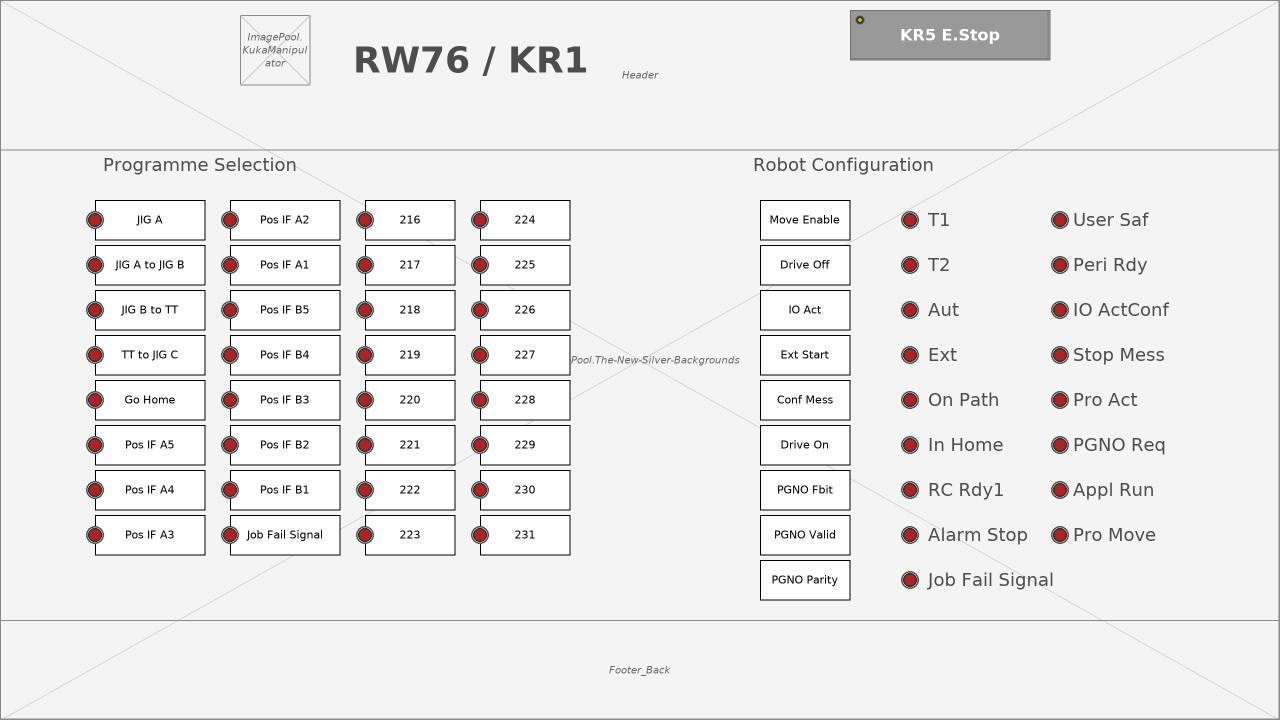
VISUALIZATION PAGE_KR5  // 1280x720
    Image (0,0 1280x720), image: ImagePool.The-New-Silver-Backgrounds
    Frame (0,620 1280x100)
        shows Footer_Back()
    Frame (0,0 1280x150)
        shows Header()
    Label (350,40 300x40), "RW76 / KR1"
    Label (100,150 200x30), "Programme Selection"
    Label (750,150 200x30), "Robot Configuration"
    Lamp1 (900,210 20x20), variable: KR5.bInBit[1,0], style: Lamp-Lamp1-Red
    Lamp1 (900,255 20x20), variable: KR5.bInBit[1,1], style: Lamp-Lamp1-Red
    Lamp1 (900,300 20x20), variable: KR5.bInBit[1,2], style: Lamp-Lamp1-Red
    Lamp1 (900,345 20x20), variable: KR5.bInBit[1,3], style: Lamp-Lamp1-Red
    Lamp1 (900,390 20x20), variable: KR5.bInBit[1,4], style: Lamp-Lamp1-Red
    Lamp1 (900,435 20x20), variable: KR5.bInBit[1,5], style: Lamp-Lamp1-Red
    Lamp1 (900,480 20x20), variable: KR5.bInBit[1,6], style: Lamp-Lamp1-Red
    Lamp1 (900,525 20x20), variable: KR5.bInBit[1,7], style: Lamp-Lamp1-Red
    Lamp1 (1050,210 20x20), variable: KR5.bInBit[2,0], style: Lamp-Lamp1-Red
    Lamp1 (1050,255 20x20), variable: KR5.bInBit[2,1], style: Lamp-Lamp1-Red
    Lamp1 (1050,300 20x20), variable: KR5.bInBit[2,2], style: Lamp-Lamp1-Red
    Lamp1 (1050,345 20x20), variable: KR5.bInBit[2,3], style: Lamp-Lamp1-Red
    Lamp1 (1050,390 20x20), variable: KR5.bInBit[2,4], style: Lamp-Lamp1-Red
    Lamp1 (1050,435 20x20), variable: KR5.bInBit[2,5], style: Lamp-Lamp1-Red
    Lamp1 (1050,480 20x20), variable: KR5.bInBit[2,6], style: Lamp-Lamp1-Red
    Lamp1 (1050,525 20x20), variable: KR5.bInBit[2,7], style: Lamp-Lamp1-Red
    Group (850,10 200x50)
        Button (0,0 200x50), "KR5 E.Stop"
            toggle KR5.KR5_Estop
        Lamp1 (5,5 10x10), variable: KR5.KR5_Estop, style: Lamp-Lamp1-Yellow
    Image (240,15 70x70), image: ImagePool.KukaManipulator
    RoundedRectangle (760,200 90x40), "Move Enable"
        toggle KR5.bOutBit[1,0]
    RoundedRectangle (760,245 90x40), "Drive Off"
        toggle KR5.bOutBit[1,1]
    RoundedRectangle (760,290 90x40), "IO Act"
        toggle KR5.bOutBit[1,2]
    RoundedRectangle (760,335 90x40), "Ext Start"
        toggle KR5.bOutBit[1,3]
    RoundedRectangle (760,380 90x40), "Conf Mess"
        toggle KR5.bOutBit[1,4]
    RoundedRectangle (760,425 90x40), "Drive On"
        toggle KR5.bOutBit[1,5]
    RoundedRectangle (760,470 90x40), "PGNO Fbit"
        toggle KR5.bOutBit[1,6]
    RoundedRectangle (760,515 90x40), "PGNO Valid"
        toggle KR5.bOutBit[1,7]
    RoundedRectangle (760,560 90x40), "PGNO Parity"
        toggle KR5.bOutBit[2,0]
    RoundedRectangle (95,200 110x40), "JIG A"
        toggle KR5.bOutBit[3,0]
    RoundedRectangle (95,245 110x40), "JIG A to JIG B"
        toggle KR5.bOutBit[3,1]
    RoundedRectangle (95,290 110x40), "JIG B to TT"
        toggle KR5.bOutBit[3,2]
    RoundedRectangle (95,335 110x40), "TT to JIG C"
        toggle KR5.bOutBit[3,3]
    RoundedRectangle (95,380 110x40), "Go Home"
        toggle KR5.bOutBit[3,4]
    RoundedRectangle (95,425 110x40), "Pos IF A5"
        toggle KR5.bOutBit[3,5]
    RoundedRectangle (95,470 110x40), "Pos IF A4"
        toggle KR5.bOutBit[3,6]
    RoundedRectangle (95,515 110x40), "Pos IF A3"
        toggle KR5.bOutBit[3,7]
    Label (1070,205 110x30), "User Saf"
    Label (1070,250 110x30), "Peri Rdy"
    Label (1070,295 110x30), "IO ActConf"
    Label (1070,340 110x30), "Stop Mess"
    Label (1070,385 110x30), "Pro Act"
    Label (1070,430 110x30), "PGNO Req"
    Label (1070,475 110x30), "Appl Run"
    Label (1070,520 110x30), "Pro Move"
    Label (925,205 105x30), "T1"
    Label (925,250 105x30), "T2"
    Label (925,295 105x30), "Aut"
    Label (925,340 105x30), "Ext"
    Label (925,385 105x30), "On Path"
    Label (925,430 105x30), "In Home"
    Label (925,475 105x30), "RC Rdy1"
    Label (925,520 105x30), "Alarm Stop"
    Label (925,565 200x30), "Job Fail Signal"
    Lamp1 (900,570 20x20), variable: KR5.bInBit[4,7], style: Lamp-Lamp1-Red
    RoundedRectangle (230,200 110x40), "Pos IF A2"
        toggle KR5.bOutBit[4,0]
    RoundedRectangle (230,245 110x40), "Pos IF A1"
        toggle KR5.bOutBit[4,1]
    RoundedRectangle (230,290 110x40), "Pos IF B5"
        toggle KR5.bOutBit[4,2]
    RoundedRectangle (230,335 110x40), "Pos IF B4"
        toggle KR5.bOutBit[4,3]
    RoundedRectangle (230,380 110x40), "Pos IF B3"
        toggle KR5.bOutBit[4,4]
    RoundedRectangle (230,425 110x40), "Pos IF B2"
        toggle KR5.bOutBit[4,5]
    RoundedRectangle (230,470 110x40), "Pos IF B1"
        toggle KR5.bOutBit[4,6]
    RoundedRectangle (230,515 110x40), "Job Fail Signal"
        toggle KR5.bOutBit[4,7]
    RoundedRectangle (480,200 90x40), "224"
        toggle KR5.bOutBit[6,0]
    RoundedRectangle (480,245 90x40), "225"
        toggle KR5.bOutBit[6,1]
    RoundedRectangle (480,290 90x40), "226"
        toggle KR5.bOutBit[6,2]
    RoundedRectangle (480,335 90x40), "227"
        toggle KR5.bOutBit[6,3]
    RoundedRectangle (480,380 90x40), "228"
        toggle KR5.bOutBit[6,4]
    RoundedRectangle (480,425 90x40), "229"
        toggle KR5.bOutBit[6,5]
    RoundedRectangle (480,470 90x40), "230"
        toggle KR5.bOutBit[6,6]
    RoundedRectangle (480,515 90x40), "231"
        toggle KR5.bOutBit[6,7]
    Lamp1 (470,210 20x20), variable: KR5.bInBit[6,0], style: Lamp-Lamp1-Red
    Lamp1 (470,255 20x20), variable: KR5.bInBit[6,1], style: Lamp-Lamp1-Red
    Lamp1 (470,300 20x20), variable: KR5.bInBit[6,2], style: Lamp-Lamp1-Red
    Lamp1 (470,345 20x20), variable: KR5.bInBit[6,3], style: Lamp-Lamp1-Red
    Lamp1 (470,390 20x20), variable: KR5.bInBit[6,4], style: Lamp-Lamp1-Red
    Lamp1 (470,435 20x20), variable: KR5.bInBit[6,5], style: Lamp-Lamp1-Red
    Lamp1 (470,480 20x20), variable: KR5.bInBit[6,6], style: Lamp-Lamp1-Red
    Lamp1 (470,525 20x20), variable: KR5.bInBit[6,7], style: Lamp-Lamp1-Red
    RoundedRectangle (365,200 90x40), "216"
        toggle KR5.bOutBit[5,0]
    RoundedRectangle (365,245 90x40), "217"
        toggle KR5.bOutBit[5,1]
    RoundedRectangle (365,290 90x40), "218"
        toggle KR5.bOutBit[5,2]
    RoundedRectangle (365,335 90x40), "219"
        toggle KR5.bOutBit[5,3]
    RoundedRectangle (365,380 90x40), "220"
        toggle KR5.bOutBit[5,4]
    RoundedRectangle (365,425 90x40), "221"
        toggle KR5.bOutBit[5,5]
    RoundedRectangle (365,470 90x40), "222"
        toggle KR5.bOutBit[5,6]
    RoundedRectangle (365,515 90x40), "223"
        toggle KR5.bOutBit[5,7]
    Lamp1 (355,210 20x20), variable: KR5.bInBit[5,0], style: Lamp-Lamp1-Red
    Lamp1 (355,255 20x20), variable: KR5.bInBit[5,1], style: Lamp-Lamp1-Red
    Lamp1 (355,300 20x20), variable: KR5.bInBit[5,2], style: Lamp-Lamp1-Red
    Lamp1 (355,345 20x20), variable: KR5.bInBit[5,3], style: Lamp-Lamp1-Red
    Lamp1 (355,390 20x20), variable: KR5.bInBit[5,4], style: Lamp-Lamp1-Red
    Lamp1 (355,435 20x20), variable: KR5.bInBit[5,5], style: Lamp-Lamp1-Red
    Lamp1 (355,480 20x20), variable: KR5.bInBit[5,6], style: Lamp-Lamp1-Red
    Lamp1 (355,525 20x20), variable: KR5.bInBit[5,7], style: Lamp-Lamp1-Red
    Lamp1 (220,210 20x20), variable: KR5.bInBit[4,0], style: Lamp-Lamp1-Red
    Lamp1 (220,255 20x20), variable: KR5.bInBit[4,1], style: Lamp-Lamp1-Red
    Lamp1 (220,300 20x20), variable: KR5.bInBit[4,2], style: Lamp-Lamp1-Red
    Lamp1 (220,345 20x20), variable: KR5.bInBit[4,3], style: Lamp-Lamp1-Red
    Lamp1 (220,390 20x20), variable: KR5.bInBit[4,4], style: Lamp-Lamp1-Red
    Lamp1 (220,435 20x20), variable: KR5.bInBit[4,5], style: Lamp-Lamp1-Red
    Lamp1 (220,480 20x20), variable: KR5.bInBit[4,6], style: Lamp-Lamp1-Red
    Lamp1 (220,525 20x20), variable: KR5.bInBit[4,7], style: Lamp-Lamp1-Red
    Lamp1 (85,210 20x20), variable: KR5.bInBit[3,0], style: Lamp-Lamp1-Red
    Lamp1 (85,255 20x20), variable: KR5.bInBit[3,1], style: Lamp-Lamp1-Red
    Lamp1 (85,300 20x20), variable: KR5.bInBit[3,2], style: Lamp-Lamp1-Red
    Lamp1 (85,345 20x20), variable: KR5.bInBit[3,3], style: Lamp-Lamp1-Red
    Lamp1 (85,390 20x20), variable: KR5.bInBit[3,4], style: Lamp-Lamp1-Red
    Lamp1 (85,435 20x20), variable: KR5.bInBit[3,5], style: Lamp-Lamp1-Red
    Lamp1 (85,480 20x20), variable: KR5.bInBit[3,6], style: Lamp-Lamp1-Red
    Lamp1 (85,525 20x20), variable: KR5.bInBit[3,7], style: Lamp-Lamp1-Red
END_VISUALIZATION

(* stored: Version 1.1.0.1, ProductVersion 3.1.4024.12
   Visu PAGE_KR5: Id {670d242a-d394-49d8-a732-c867da6c3071} *)
